{attribute 'GeneratedUsingTerminal: EK1100-0000-0018'}
{attribute addProperty BoxType "EK1100-0000-0018"}
{attribute addProperty Id "Beckhoff_EP2xxxEK1122Beckhoff_EP2xxxEK1122_471DEECD3266"}
{attribute addProperty CRC "646026951"}
{attribute addProperty Size "3266"}
TYPE Beckhoff_EP2xxx_268196C7 EXTENDS EK1100_1FC0878B :
STRUCT
	{attribute addProperty Name "Beckhoff_EP2xxxEK1122"}
	{attribute addProperty PreviousPort "Beckhoff EP2xxx : B"}
	Beckhoff_EP2xxxEK1122 : Beckhoff_EP2xxxEK1122_471DEECD;
END_STRUCT
END_TYPE

(* stored: Version 1.2.0.0, ProductVersion 3.1.4024.9
   DUT Beckhoff_EP2xxx_268196C7: Id {5ea052d5-8e17-467e-8814-d249b66fa9c7} *)
